INTERFACE I_TestResultLogger

METHOD PUBLIC LogTestSuiteResults
VAR_INPUT
    TestResults : REFERENCE TO ARRAY[1..GVL_Param_TcUnit.MaxNumberOfTestSuites] OF ST_TestSuiteResult;
END_VAR
END_METHOD

END_INTERFACE

(* stored: Version 1.1.0.1, ProductVersion 3.1.4022.18
   Itf I_TestResultLogger: Id {fa75ee61-43fb-4767-8061-125a3a9e3424}
   Method LogTestSuiteResults: Id {033e8873-ad7a-489b-8ba9-f0de8a344939} *)
